Fanuc KAREL source: kx00020.KL

-- PROVISIONAL review KL for V770-1; original PC SHA256 ff94feebc02f210a25ef22ea26cfab9eb6a1737fb047eb2921da4a6b7a542da3
-- Incomplete behavior may be omitted. Consult companion uncertainty JSON. Do not deploy.
PROGRAM KX00020
%NOLOCKGROUP
BEGIN
  -- UNRESOLVED_PC offsets 5-17; opcodes 3F,22,9D,33,61
  -- UNRESOLVED_PC offsets 22-37; opcodes 22,9D,33,5E,75
  -- UNRESOLVED_PC offsets 42-46; opcodes 7F
END KX00020
